{region '#Template'}
	{attribute 'Version' := '5.0.1.0'}
	{attribute 'Tags' := '"LCID": "1031", "Text": "AC, Aggregates, Cooler, Temperature, Controller"'}
	{attribute 'Tags' := '"LCID": "1033", "Text": "AC, Aggregates, Cooler, Temperature, Controller"'}
	{attribute 'Using' := '"Type": "Template", "URI": "BA2_Param"'}
	{attribute 'Using' := '"Type": "Template", "URI": "EC_ID"'}
	{attribute 'Using' := '"Type": "Template", "URI": "E_BA_AC_SeqNumber_T"'}
	{attribute 'Description' := '"LCID": "1031", "Text": "Kühler Zuluft Regler Temperatur"'}
	{attribute 'Description' := '"LCID": "1033", "Text": "Cooler Supply air controller temperature"'}
{endregion}
FUNCTION_BLOCK FB_BA_AC_ColTSuACtrl EXTENDS FB_BA_View
VAR_INPUT
	bEn						: BOOL;
	fSpTSuA					: REAL;// Sollwert Temperatur kühlen // Setpoint temperature cooling
	fTSuA					: REAL;// Zuluft Temperatur // Supply air temperature
	bSync					: BOOL;
	fSync					: REAL;
END_VAR
VAR_OUTPUT
	fY              		: REAL;
	bIsActive				: BOOL;	//	active sequence controller
	bSeqActv				: BOOL;	//	Release sequence link, sequence control is active		
END_VAR
VAR_IN_OUT
	stSeqLink				: ST_BA_SeqLink;	//	Sequenz Link Struktur	//	Sequence link structure	
END_VAR
VAR_INPUT CONSTANT
	Ctrl					: FB_BA_SeqCtrl;
END_VAR

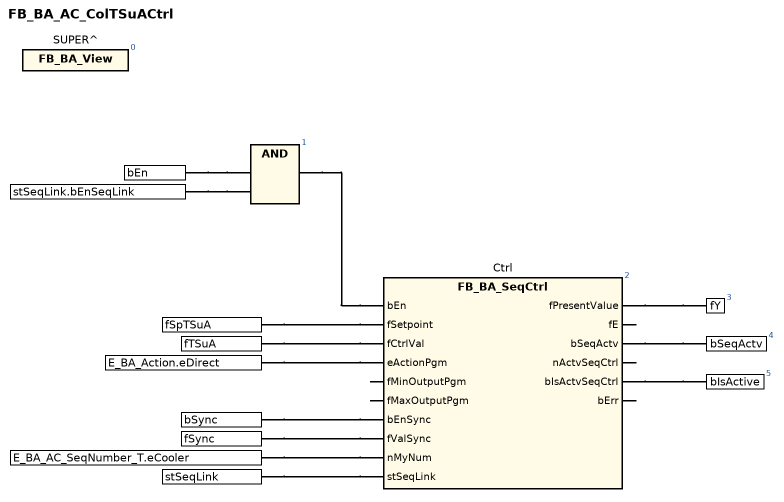
SUPER^(); // FB_BA_View
Ctrl(
    bEn := bEn AND stSeqLink.bEnSeqLink,
    fSetpoint := fSpTSuA,
    fCtrlVal := fTSuA,
    eActionPgm := E_BA_Action.eDirect,
    bEnSync := bSync,
    fValSync := fSync,
    nMyNum := E_BA_AC_SeqNumber_T.eCooler,
    stSeqLink := stSeqLink); // FB_BA_SeqCtrl
fY := Ctrl.fPresentValue;
bSeqActv := Ctrl.bSeqActv;
bIsActive := Ctrl.bIsActvSeqCtrl;

METHOD FB_init : BOOL
VAR_INPUT
	bInitRetains : BOOL; // if TRUE, the retain variables are initialized (warm start / cold start)
	bInCopyCode : BOOL;  // if TRUE, the instance afterwards gets moved into the copy code (online change)
END_VAR
Ctrl.iParent						:= THIS^;
Ctrl.iLabel							:= LblFun_LoopObject; 
Ctrl.sObjectName					:= '{Idx=01}';						 
Ctrl.eOpMode						:= E_BA_PIDMode.ePID;								 	 										 	
Ctrl.eOutputUnit					:= E_BA_Unit.eOther_Percent;
Ctrl.fProportionalConstant			:= 3;
Ctrl.fIntegralConstant				:= 180;
Ctrl.fDerivativeConstant			:= 0;
Ctrl.fMaxOutputRm 					:= 100;
Ctrl.fMinOutputRm					:= 0;
Ctrl.fCOVIncrement					:= 0;
Ctrl.nDampConstant					:= 0;
Ctrl.fNeutralZone					:= 0;
END_METHOD

END_FUNCTION_BLOCK

(* stored: Version 1.1.0.1, ProductVersion 3.1.4024.12
   POU FB_BA_AC_ColTSuACtrl: Id {00f77247-410d-4136-a871-d54a2156b99a}, SpecialFunc None
   Method FB_init: Id {d7d20e92-4553-4504-9685-492b4e0687c5} *)
